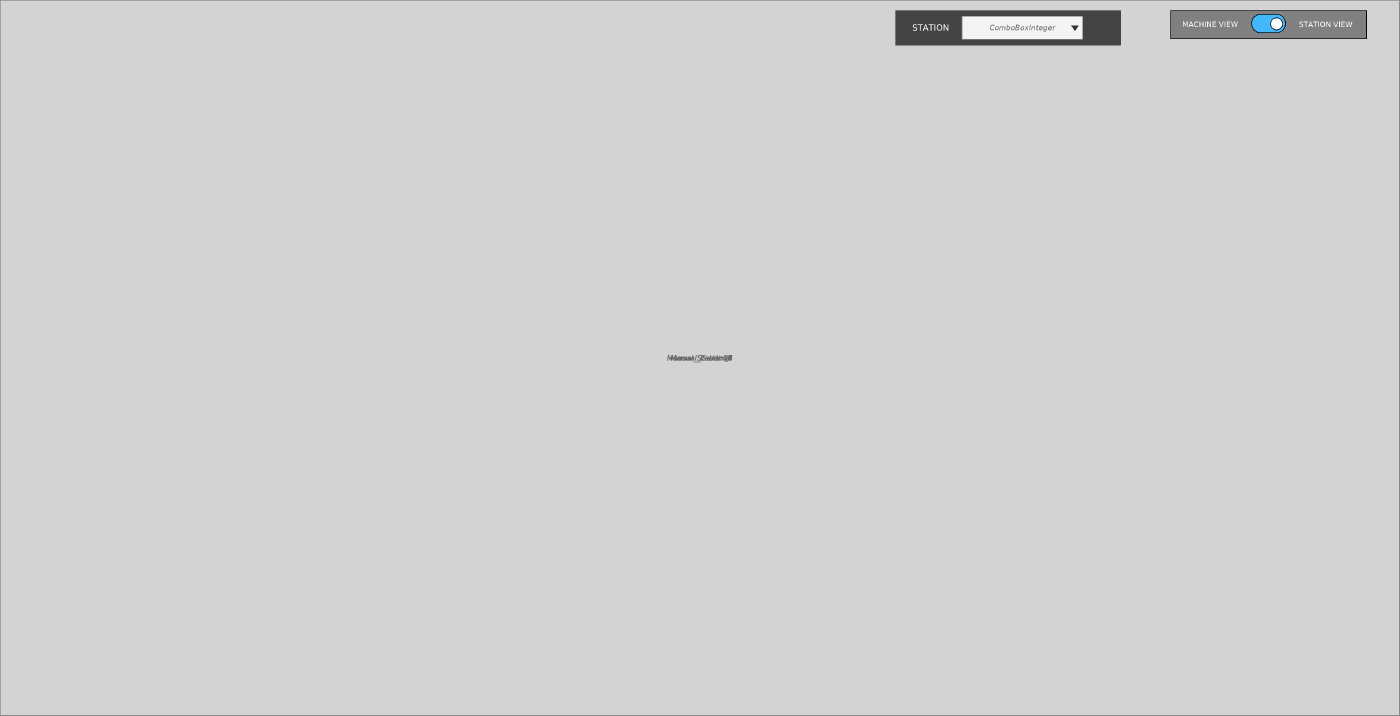
VISUALIZATION Manual_AllStation  // 1920x983
    Rectangle (0,0 1920x983)
    Frame (0,0 1920x983), invisible if: HMI_Ctrl.StationInfoPageNo <> 1
        shows Manual_Station01()
    Frame (0,0 1920x983), invisible if: HMI_Ctrl.StationInfoPageNo <> 2
        shows Manual_Station02()
    Frame (0,0 1920x983), invisible if: HMI_Ctrl.StationInfoPageNo <> 3
        shows Manual_Station03()
    Frame (0,0 1920x983), invisible if: HMI_Ctrl.StationInfoPageNo <> 4
        shows Manual_Station04()
    Frame (0,0 1920x983), invisible if: HMI_Ctrl.StationInfoPageNo <> 5
        shows Manual_Station05()
    Frame (0,0 1920x983), invisible if: HMI_Ctrl.StationInfoPageNo <> 6
        shows Manual_Station06()
    Frame (0,0 1920x983), invisible if: HMI_Ctrl.StationInfoPageNo <> 7
        shows Manual_Loading()
    Frame (0,0 1920x983), invisible if: HMI_Ctrl.StationInfoPageNo <> 0
        shows Manual_General()
    Group (1605,13 269x41)
        RoundedRectangle (0,1 269x39)
        Label (1,0 108x41), "MACHINE VIEW"
        Label (161,0 105x41), "STATION VIEW"
        Group (111,6 47x26)
            OnMouseClick: toggle HMI_Ctrl.AutoStationViewEnable
            Ellipse (0,0 26x26)
            Ellipse (21,0 26x26)
            RoundedRectangle (8,0 29x26)
            Ellipse (1,1 24x24)
            Ellipse (23,1 23x24)
            RoundedRectangle (9,1 28x24)
            Ellipse (26,5 17x17)
    Group (1228,14 272x48)
        RoundedRectangle (0,0 309x48)
        Label (20,12 79x24), "STATION"
    ComboBoxInteger (1319,22 166x32), variable: HMI_Ctrl.StationInfoPageNo, invisible if: NOT HMI_Ctrl.AutoStationViewEnable, text list: 'TextList_ManualPage'
END_VISUALIZATION

(* stored: Version 1.1.0.1, ProductVersion 3.1.4024.12
   Visu Manual_AllStation: Id {94ef6030-e771-479a-91d5-17f409511f62} *)
